// Abstract base for TcForge device-like function blocks. Provides:
//   - built-in fault book-keeping (current + last + persistent ring buffer)
//   - the source-lock flag (bSourceLockedToProg)
//   - safety-command primitives (Reset) that are always accepted
//   - diagnostics methods (IsFaulted / GetFaultCode / GetFaultString)
//   - protected helpers for children to populate ST_DeviceHeader_Sts
//
// Children:
//   - EXTEND this FB and declare their own sts containing ST_DeviceHeader_Sts
//     as the first member named `header`
//   - override ResolveFaultString(code) to map their device-specific fault
//     enum to human-readable text
//   - call _Raise(code, source, reason) to register a fault (idempotent on
//     `code`); _ClearFault() to clear without losing history
//   - call _AcceptCommand(eRequester) at the end of every accepted method
//   - call _UpdateHeader(sts.header, ...) once per cycle from the body
//
// Fault semantics:
//   - _Raise is idempotent on `code`. Repeated calls with the same non-zero
//     code push only one ring entry per episode; a different code replaces
//     the current fault and pushes a new entry (so a progression like
//     Timeout -> OddStep is preserved).
//   - _ClearFault wipes the active fault only. last* fields and the ring
//     survive so HMIs can still show what happened.
//   - The last-fault fields and ring buffer are PERSISTENT so that a process
//     restart does not silently lose the most recent fault context.
FUNCTION_BLOCK ABSTRACT FB_DeviceBase
VAR CONSTANT
    FAULT_RING_SIZE : UDINT := 8;
END_VAR

VAR
    {attribute 'OPC.UA.DA' := '0'}
    _operatorMailbox : FB_OperatorMailbox;
    {attribute 'OPC.UA.DA' := '0'}
    bSourceLockedToProg : BOOL;
    {attribute 'OPC.UA.DA' := '0'}
    _lastRequester : E_Requester;
    {attribute 'OPC.UA.DA' := '0'}
    _tsLastCommand : LTIME;

    // Active fault (not persistent; Reset on restart so recovery logic re-runs).
    {attribute 'OPC.UA.DA' := '0'}
    _faultCode   : DINT;
    {attribute 'OPC.UA.DA' := '0'}
    _faultTs     : LTIME;
    {attribute 'OPC.UA.DA' := '0'}
    _faultSource : STRING(31);
    {attribute 'OPC.UA.DA' := '0'}
    _faultReason : STRING(79);
END_VAR

VAR PERSISTENT
    // Most recent fault — survives Reset (and PLC restart) so HMIs can always
    // show "last fault info".
    _lastFaultCode      : DINT;
    _lastFaultTs        : LTIME;
    _lastFaultRequester : E_Requester;
    _lastFaultSource    : STRING(31);
    _lastFaultReason    : STRING(79);

    // Short ring-buffer history.
    _faultRing     : ARRAY[0..7] OF ST_FaultEntry;
    _faultRingHead : UDINT;
END_VAR

// Abstract base — children implement their own cyclic logic.

// Base Reset clears diagnostics from any requester, regardless
// of source lock or current fault state. Clears the active fault; history is
// preserved in the ring buffer. Children may override to add device-specific
// recovery validation and cleanup. Successful overrides call SUPER^.Reset;
// the state machine rejects Reset until STOPPED and running conditions are good.
METHOD PUBLIC Reset : E_RpcMethodResponse
VAR_INPUT
    eRequester : E_Requester := E_Requester.PROG;
END_VAR
// Reject invalid identity before any command-specific mutation.
Reset := F_ValidateRequester(eRequester := eRequester, bSourceLocked := FALSE, bFaulted := FALSE);
IF Reset <> E_RpcMethodResponse.ACCEPTED THEN RETURN; END_IF;
_operatorMailbox.CancelNormal();
_ClearFault();
_AcceptCommand(eRequester := eRequester);
Reset := E_RpcMethodResponse.ACCEPTED;
END_METHOD

METHOD PUBLIC LockSource : E_RpcMethodResponse
VAR_INPUT
    bLock : BOOL;
END_VAR
bSourceLockedToProg := bLock;
LockSource := E_RpcMethodResponse.ACCEPTED;
END_METHOD

METHOD PUBLIC IsFaulted : BOOL
IsFaulted := _faultCode <> 0;
END_METHOD

METHOD PUBLIC GetFaultCode : DINT
GetFaultCode := _faultCode;
END_METHOD

METHOD PUBLIC GetFaultString : STRING(79)
// Virtual dispatch: child's ResolveFaultString() maps the current code.
GetFaultString := THIS^.ResolveFaultString(code := _faultCode);
END_METHOD

// Children override to translate their fault-enum value into human-readable
// text. Default returns empty so devices without a fault model still compile.
METHOD PROTECTED ResolveFaultString : STRING(79)
VAR_INPUT
    code : DINT;
END_VAR
ResolveFaultString := '';
END_METHOD

// Book-keeping called at the end of every accepted command method.
METHOD PROTECTED _AcceptCommand
VAR_INPUT
    eRequester : E_Requester;
END_VAR
_lastRequester := eRequester;
_tsLastCommand := F_Now();
END_METHOD

// Raise a fault with optional source (where it came from) and reason (free-form).
// Idempotent on `code`: a second call with the same non-zero code in the
// same episode is a no-op (returns FALSE) even if source/reason differ — so
// cyclic callers can spam this without flooding the ring. A different
// non-zero code replaces the current fault and pushes a new ring entry.
// The requester recorded with the fault is the most recent command requester
// (_lastRequester), which is what the operator / HMI has context for.
// Returns TRUE when a new ring entry was pushed this call.
METHOD PROTECTED _Raise : BOOL
VAR_INPUT
    code   : DINT;
    source : STRING(31);
    reason : STRING(79);
END_VAR
IF code = 0 THEN
    _Raise := FALSE;
    RETURN;
END_IF;

IF code = _faultCode THEN
    _Raise := FALSE;
    RETURN;
END_IF;

_faultCode   := code;
_faultTs     := F_Now();
_faultSource := source;
_faultReason := reason;

_lastFaultCode      := code;
_lastFaultTs        := _faultTs;
_lastFaultRequester := _lastRequester;
_lastFaultSource    := source;
_lastFaultReason    := reason;

_faultRingHead := _faultRingHead MOD FAULT_RING_SIZE;
_faultRing[_faultRingHead].code      := code;
_faultRing[_faultRingHead].ts        := _faultTs;
_faultRing[_faultRingHead].requester := _lastRequester;
_faultRing[_faultRingHead].source    := source;
_faultRing[_faultRingHead].reason    := reason;
_faultRingHead := (_faultRingHead + 1) MOD FAULT_RING_SIZE;

_Raise := TRUE;
END_METHOD

// Clear the currently-active fault. Preserves the ring buffer and the
// last-fault fields so HMIs can still show what happened.
METHOD PROTECTED _ClearFault
_faultCode   := 0;
_faultTs     := LTIME#0ns;
_faultSource := '';
_faultReason := '';
END_METHOD

// Refreshes the common header a child embeds as `header` in its sts struct.
// Call once per cycle from the child's cyclic body. Device-specific fields
// (advanced, value, etc.) stay in the child sts alongside `header`.
METHOD PROTECTED _UpdateHeader
VAR_IN_OUT
    header : ST_DeviceHeader_Sts;
END_VAR
VAR_INPUT
    stateString : STRING(31);
    busy     : BOOL;
END_VAR
header.stateString     := stateString;
header.busy         := busy;
header.faulted      := _faultCode <> 0;
header.ready        := NOT header.faulted AND NOT busy AND NOT bSourceLockedToProg;
header.sourceLocked := bSourceLockedToProg;
header.faultCode       := _faultCode;
header.faultString     := THIS^.ResolveFaultString(code := _faultCode);
header.faultSource     := _faultSource;
header.faultReason     := _faultReason;
header.lastFaultCode   := _lastFaultCode;
header.lastFaultString := THIS^.ResolveFaultString(code := _lastFaultCode);
header.lastFaultSource := _lastFaultSource;
header.lastFaultReason := _lastFaultReason;
header.lastRequester   := _lastRequester;
header.tsLastCommand   := _tsLastCommand;
header.tsLastFault     := _lastFaultTs;
END_METHOD

{attribute 'TcRpcEnable' := '1'}
METHOD PUBLIC OperatorReset : E_RpcMethodResponse

VAR_INPUT requestId : ULINT; END_VAR
OperatorReset := _operatorMailbox.Submit(requestId := requestId, command := E_OperatorCommand.Reset, value := 0.0);
END_METHOD

{attribute 'TcRpcEnable' := '1'}
METHOD PUBLIC OperatorCommandResult : E_RpcMethodResponse
VAR_INPUT requestId : ULINT; END_VAR
OperatorCommandResult := _operatorMailbox.GetResult(requestId := requestId);
END_METHOD

METHOD PROTECTED _ProcessOperatorCommands
VAR command : E_OperatorCommand; value : REAL; result : E_RpcMethodResponse; END_VAR
IF _operatorMailbox.BeginConsume(command => command, value => value) THEN
    result := THIS^._DispatchOperatorCommand(command := command, value := value);
    _operatorMailbox.EndConsume(result := result);
END_IF;
END_METHOD

METHOD PROTECTED _DispatchOperatorCommand : E_RpcMethodResponse
VAR_INPUT command : E_OperatorCommand; value : REAL; END_VAR
CASE command OF
E_OperatorCommand.Reset: _DispatchOperatorCommand := THIS^.Reset(eRequester := E_Requester.OPERATOR);
ELSE _DispatchOperatorCommand := E_RpcMethodResponse.REJECTED_INVALID_PARAMETER;
END_CASE;
END_METHOD

END_FUNCTION_BLOCK

(* stored: Version 1.1.0.1, ProductVersion 3.1.4026.12
   POU FB_DeviceBase: Id {c0000001-0000-0000-0000-000000000001}, SpecialFunc None
   Folder Safety: Id {c0000001-0000-0000-f000-000000000001}
   Folder Diagnostics: Id {c0000001-0000-0000-f000-000000000002}
   Folder Protected: Id {c0000001-0000-0000-f000-000000000003}
   Method Reset: Id {c0000001-0000-0000-1000-000000000001}
   Method LockSource: Id {c0000001-0000-0000-1000-000000000002}
   Method IsFaulted: Id {c0000001-0000-0000-1000-000000000003}
   Method GetFaultCode: Id {c0000001-0000-0000-1000-000000000004}
   Method GetFaultString: Id {c0000001-0000-0000-1000-000000000005}
   Method ResolveFaultString: Id {c0000001-0000-0000-1000-000000000006}
   Method _AcceptCommand: Id {c0000001-0000-0000-1000-000000000007}
   Method _Raise: Id {c0000001-0000-0000-1000-000000000008}
   Method _ClearFault: Id {c0000001-0000-0000-1000-000000000009}
   Method _UpdateHeader: Id {c0000001-0000-0000-1000-00000000000a}
   Method OperatorReset: Id {1ff20d7b-3ab2-48a6-b25f-458b50a21eec}
   Method OperatorCommandResult: Id {c6b8086b-4a61-471d-bc0a-5f1111c8623e}
   Method _ProcessOperatorCommands: Id {b9227d48-50f9-4f57-b40f-1adca118f38b}
   Method _DispatchOperatorCommand: Id {94fe5150-ee7b-447c-92ba-8317950b56d8} *)
